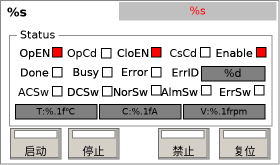
VISUALIZATION TMPModuleVisu  // 280x165
VAR_IN_OUT
	userData: TMPHMIStruts;
END_VAR
    Button (10,128 51x31), "启动", input disabled if: NOT userData.HMIEnable
        tap userData.open
    Rectangle (14,130 43x8), colour toggle: userData.openRelay
    GroupBox (9,27 263x99), "Status"
        RoundedRectangle (43,40 10x10), colour toggle: userData.done
        RoundedRectangle (247,20 10x10), colour toggle: userData.enable
        RoundedRectangle (93,40 10x10), colour toggle: userData.busy
        RoundedRectangle (142,40 10x10), colour toggle: userData.error
        Rectangle (192,39 64x15), "%d", text variable: userData.errID
        Label (7,20 37x13), "OpEN"
        RoundedRectangle (43,20 10x10), colour toggle: userData.enableOpen
        Label (106,20 37x13), "CloEN"
        RoundedRectangle (142,20 10x10), colour toggle: userData.enableClose
        Label (208,20 39x13), "Enable"
        Label (160,39 33x14), "ErrID"
        Label (112,39 30x13), "Error"
        Label (63,39 30x13), "Busy"
        Label (10,38 33x16), "Done"
        RoundedRectangle (43,59 10x10), colour toggle: userData.AccAprSw
        RoundedRectangle (93,59 10x10), colour toggle: userData.DccAprSw
        Label (56,59 37x13), "DCSw"
        Label (105,59 37x13), "NorSw"
        RoundedRectangle (142,58 10x10), colour toggle: userData.NormalAprSw
        Label (152,59 40x13), "AlmSw"
        RoundedRectangle (192,58 10x10), colour toggle: userData.AlmAprSw
        Label (208,59 37x13), "ErrSw"
        RoundedRectangle (245,58 10x10), colour toggle: userData.ErrorAprSw
        Rectangle (6,77 82x15), "T:%.1f℃", text variable: userData.temperature, input disabled if: true
        Rectangle (90,77 82x15), "C:%.1fA", text variable: userData.current, input disabled if: true
        Rectangle (174,77 82x15), "V:%.1frpm", text variable: userData.speed, input disabled if: true
        Label (157,20 34x13), "CsCd"
    RoundedRectangle (52,67 10x10), colour toggle: userData.done
    RoundedRectangle (256,47 10x10), colour toggle: userData.enable
    RoundedRectangle (102,67 10x10), colour toggle: userData.busy
    RoundedRectangle (151,67 10x10), colour toggle: userData.error
    Rectangle (201,66 64x15), "%d", text variable: userData.errID, input disabled if: true
    Label (16,47 37x13), "OpEN"
    RoundedRectangle (52,47 10x10), colour toggle: userData.enableOpen
    Label (115,47 37x13), "CloEN"
    RoundedRectangle (151,47 10x10), colour toggle: userData.enableClose
    Label (217,47 39x13), "Enable"
    Label (169,66 33x14), "ErrID"
    Label (121,66 30x13), "Error"
    Label (72,66 30x13), "Busy"
    Label (19,65 33x16), "Done"
    RoundedRectangle (52,86 10x10), colour toggle: userData.AccAprSw
    RoundedRectangle (102,86 10x10), colour toggle: userData.DccAprSw
    Label (65,86 37x13), "DCSw"
    Label (114,86 37x13), "NorSw"
    RoundedRectangle (151,85 10x10), colour toggle: userData.NormalAprSw
    Label (161,86 40x13), "AlmSw"
    RoundedRectangle (201,85 10x10), colour toggle: userData.AlmAprSw
    Label (217,86 37x13), "ErrSw"
    RoundedRectangle (254,85 10x10), colour toggle: userData.ErrorAprSw
    Button (219,128 51x31), "复位"
        tap userData.reset
    Rectangle (223,130 43x8), colour toggle: userData.resetRelay
    Rectangle (4,2 114x20), "%s", text variable: userData.nameTXT
    Button (68,128 51x31), "停止"
        tap userData.close
    Rectangle (72,130 43x8), colour toggle: userData.closeRelay
    Label (15,86 37x13), "ACSw"
    Button (158,128 51x31), "禁止"
        tap userData.stop
    Rectangle (161,130 43x8)
    Rectangle (119,2 157x18), "%s", text variable: userData.errTXT
    Label (64,47 36x13), "OpCd"
    RoundedRectangle (101,48 10x10), colour toggle: userData.opencondition
    RoundedRectangle (200,47 10x10), colour toggle: userData.closecondition
END_VISUALIZATION

(* stored: Version 1.1.0.1, ProductVersion 3.1.4024.4
   Visu TMPModuleVisu: Id {068f8943-766e-4b4e-b845-bde186cd0d17} *)
